// TIA Portal V21 export
TYPE "UDT_Device"
   STRUCT
      Mode : USInt;   // 0- Auto; 2 - Service
      Start : Bool;
      Stop : Bool;
      Reverse : Bool;
      Setpoint : Real;
      State : Int;
   END_STRUCT;
END_TYPE
